(* IEC 61131-3 sources: AXOpen/src/core/ctrl/src/AxoObject, 2 files *)

(* ---- AdamObject.st ---- *)
 NAMESPACE AXOpen.Core
    ///<summary>
    /// A root object implementation of IAxoObject to serve as an object with context but without parent.
    /// An instance of this class is used as a parent for all top-level objects in the context.
    /// It must be initialized with InitInitializeRootObject method of IAxoContext before use.
    ///</summary>
    {S7.extern=ReadWrite}
    CLASS AdamAxoObject EXTENDS AXOpen.Core.AxoObject
        VAR
            NULL_OBJECT : _NULL_OBJECT;
        END_VAR
        METHOD PUBLIC OVERRIDE GetParent : IAxoObject
            GetParent := NULL_OBJECT;
        END_METHOD
    END_CLASS
END_NAMESPACE

(* ---- AxoObject.st ---- *)
USING AXOpen.Messaging.Static;
USING AXOpen.Rtc;

NAMESPACE AXOpen.Core
    ///<summary>
    /// Provides base class for all classes of `AXOpen`.
    ///</summary>
    {S7.extern=ReadWrite}
    CLASS PUBLIC AxoObject IMPLEMENTS IAxoObject
        VAR PUBLIC
            {#ix-attr:[CompilerOmits("POCO")]}
            {#ix-attr:[IgnoreOnPocoOperation()]}
            {#ix-attr:[RenderIgnore()]}
            Identity   : ULINT := ULINT#0;

            {#ix-attr:[CompilerOmits("POCO")]}
            {#ix-attr:[IgnoreOnPocoOperation()]}
            {#ix-attr:[RenderIgnore()]}
            MsgCnt   : LINT := LINT#0;

            {#ix-attr:[CompilerOmits("POCO")]}
            {#ix-attr:[IgnoreOnPocoOperation()]}
            {#ix-attr:[RenderIgnore()]}
            {#ix-attr:[ReadOnly()]}
            _dg_   : BYTE;
        END_VAR

        VAR PRIVATE
            _parent         : IAxoObject;
            _context        : IAxoContext;
            _isInitialized  : BOOL;
            _errorState     : UINT;
        END_VAR

        VAR PRIVATE
            {#ix-attr:[CompilerOmits()]}
            {S7.extern=Hidden}
            NULL_CONTEXT : _NULL_CONTEXT;
            {#ix-attr:[CompilerOmits()]}
            {S7.extern=Hidden}
            NULL_OBJECT : _NULL_OBJECT;
        END_VAR

        ///<summary>
        /// Gets unique identity of this object in given context.
        ///</summary>
        METHOD PUBLIC GetIdentity : ULINT
            GetIdentity := Identity;
        END_METHOD

        ///<summary>
        /// Gets context in which this object was initialized.
        ///</summary>
        METHOD PUBLIC GetContext : IAxoContext
            IF(_context <> NULL) THEN
                GetContext := _context;
                _dg_.%X0 := FALSE;
            ELSE
                _dg_.%X0 := TRUE;
                GetContext := NULL_CONTEXT;
            END_IF;
        END_METHOD

        ///<summary>
        /// Gets context in which this object was initialized.
        ///</summary>
        METHOD PUBLIC GetContextUnsafe : IAxoContext
            GetContextUnsafe := _context;
        END_METHOD

        ///<summary>
        /// Gets inParent in which this object was initialized.
        ///</summary>
        METHOD PUBLIC GetParent : IAxoObject
            IF(_parent <> NULL) THEN
                GetParent := _parent;
                _dg_.%X1 := FALSE;
            ELSE
                _dg_.%X1 := TRUE;
                GetParent := NULL_OBJECT;
            END_IF;
        END_METHOD

        ///<summary>
        /// Initializes this object associating it given inParent.
        /// This method should be called only once upon the program start.
        /// Any subsequent call are ignored.
        ///</summary>
        METHOD PRIVATE Initialize
            VAR_INPUT
                inParent : IAxoObject;
            END_VAR

            VAR
                NULL_CONTEXT_OBJ    : IAxoObject;
            END_VAR

            // We always reset message count upon initialization.
            THIS.MsgCnt := _msgCntAcc;
            _msgCntAcc := LINT#0;

            IF _isInitialized THEN
                RETURN;
            END_IF;

            IF(inParent = NULL) THEN
                // TODO provide some message
                _errorState := UINT#20;
                RETURN;
            END_IF;

            NULL_CONTEXT_OBJ ?= NULL_CONTEXT;
            IF(inParent.GetContext() = NULL_CONTEXT_OBJ) THEN
                // TODO provide some message
                _errorState := UINT#30;
                RETURN;
            END_IF;

            IF(inParent = _parent) THEN
                // TODO provide some message
                _errorState := UINT#40;
                RETURN;
            END_IF;

            _context        := inParent.GetContext();
            _parent         := inParent;
            _isInitialized  := TRUE;

        END_METHOD

        METHOD PUBLIC Run
            VAR_INPUT
                inParent : IAxoObject;
            END_VAR
            THIS.Initialize(inParent);
        END_METHOD

        ///<summary>
        /// Initializes this object associating it given context.
        /// This method should be called only once upon the program start.
        /// Any subsequent call are ignored.
        ///</summary>
        METHOD INTERNAL InitializeWithContext
            VAR_INPUT
                inContext : IAxoContext;
            END_VAR

            // We always reset message count upon initialization.
            THIS.MsgCnt := _msgCntAcc;
            _msgCntAcc := LINT#0;

            IF _isInitialized THEN
                RETURN;
            END_IF;

            IF(inContext = NULL) THEN
                // TODO provide some message
                _errorState := UINT#10;
                RETURN;
            END_IF;

            _context        := inContext;
            _isInitialized  := TRUE;

        END_METHOD

        VAR PROTECTED
            {#ix-attr:[RenderIgnore()]}
            _lastMessageAggregationCycle : ULINT;
             {#ix-attr:[RenderIgnore()]}
            _msgCntAcc : LINT;
        END_VAR

        ///<summary>
        /// Aggregates message count for this object and all inParent objects in the generation of this object.
        ///</summary>
        METHOD PUBLIC AggregateMessage
            VAR_INPUT
                inCount : LINT;
            END_VAR

            IF(_context = NULL) THEN
                _context := THIS.GetContext();
                // RETURN;
            END_IF;

            IF(_lastMessageAggregationCycle <> _context.OpenCycleCount()) THEN
                THIS._msgCntAcc := LINT#0;
            END_IF;

            IF(inCount = 0) THEN
                IF(_parent <> NULL && THIS._parent <> THIS._parent.GetParent()) THEN
                    THIS._parent.AggregateMessage(inCount);
                END_IF;
                RETURN;
            END_IF;

            THIS._msgCntAcc := inCount + THIS._msgCntAcc;

            IF(_parent <> NULL && THIS._parent <> THIS._parent.GetParent()) THEN
                THIS._parent.AggregateMessage(inCount);
            END_IF;

            _lastMessageAggregationCycle := _context.OpenCycleCount();
        END_METHOD

        ///<summary>
        /// Gets whether this object is valid.
        ///</summary>
        METHOD PUBLIC IsValid : BOOL
            IsValid := TRUE;
        END_METHOD
    END_CLASS
END_NAMESPACE
